FUNCTION F_DT_TO_STRING : STRING
VAR_INPUT
	dtTime			: DT;
END_VAR
VAR
	timeStruct		: TIMESTRUCT;
END_VAR

F_DT_TO_STRING := SYSTEMTIME_TO_STRING(DT_TO_SYSTEMTIME(dtTime));

//F_DT_TO_STRING := CONCAT6(F_TO_STRING(timeStruct.wDay), '.', F_TO_STRING(timeStruct.wMonth), '.', F_TO_STRING(timeStruct.wYear), ' - ');
//F_DT_TO_STRING := CONCAT6(F_DT_TO_STRING, F_TO_STRING(timeStruct.wHour), ':', F_TO_STRING(timeStruct.wMinute), ':', F_TO_STRING(timeStruct.wSecond));

END_FUNCTION

(* stored: Version 1.1.0.1
   POU F_DT_TO_STRING: Id {0e1b1c73-5746-4a57-be3e-614719d9d625}, SpecialFunc None *)
